# EPICS StreamDevice protocol: ipApp/Db/Protura_P201.proto
InTerminator = CR;
OutTerminator = ;

ReplyTimeout = 1000;

getPos {
   out "?";
   in  "%\$1b%*s";
}
